FUNCTION_BLOCK TestLogHelper
VAR_GENERIC CONSTANT
	SubSize : USINT;
END_VAR
 EXTENDS LogHelper<SubSize>
VAR
END_VAR

METHOD GetLoggerAtIndex : I_Logger
VAR_INPUT
	Index : UDINT;
END_VAR
GetLoggerAtIndex := _SubscribedLoggers[Index];
END_METHOD

PROPERTY SubscribedCount : UDINT
GET
SubscribedCount := SubscriberCount;
END_GET
END_PROPERTY

END_FUNCTION_BLOCK

(* stored: Version 1.1.0.1, ProductVersion 3.1.4026.18
   POU TestLogHelper: Id {bf6c6d90-387c-4ae8-af46-3138d7ac899d}, SpecialFunc None
   Method GetLoggerAtIndex: Id {e18be55b-c63d-4206-bcf3-f12bd0b6bbf4}
   Property SubscribedCount: Id {c0c3bbd1-672a-4b9b-a6ec-2c27a7c8f8b2}
   Get Get: Id {60db6be2-47b7-4cce-b0ce-7258338bae32} *)
